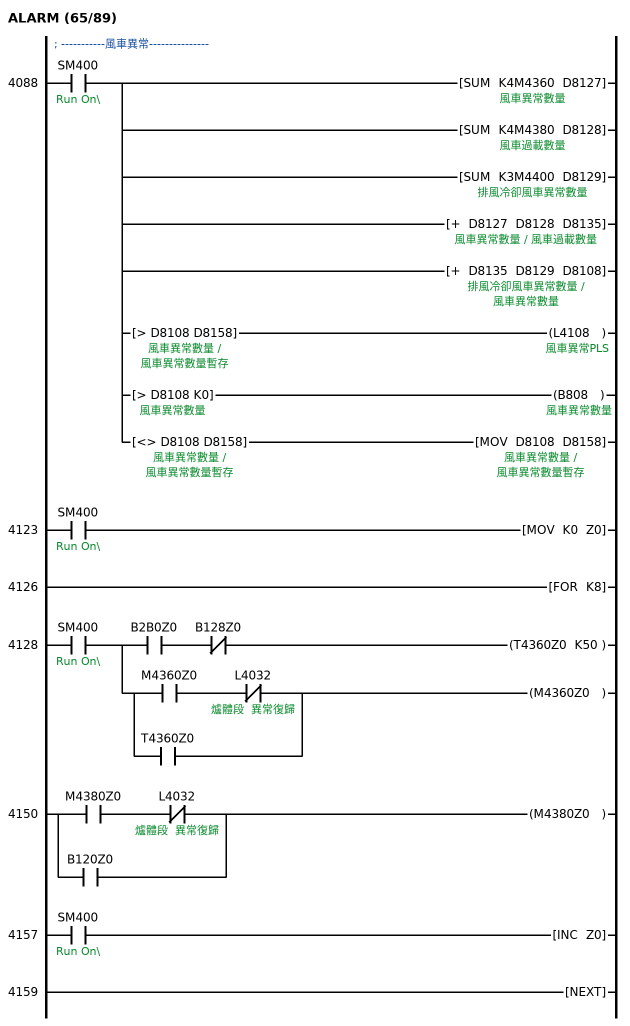
[picture p240: ladder of ALARM, rungs at steps 4088 to 4159]
; -----------風車異常---------------
4088  LD      SM400  ; Run On\
      SUM     K4M4360 D8127  ; 第01槽  風車馬達異常 / 風車異常數量
      SUM     K4M4380 D8128  ; 第01槽  風車馬達過載 / 風車過載數量
      SUM     K3M4400 D8129  ; 進料輸送排氣風車異常 / 排風冷卻風車異常數量
      +       D8127 D8128 D8135
      +       D8135 D8129 D8108  ; 風車異常數量
      MPS
      AND>    D8108 D8158  ; 風車異常數量 / 風車異常數量暫存
      OUT     L4108  ; 風車異常PLS
      MRD
      AND>    D8108 K0  ; 風車異常數量
      OUT     B808  ; 風車異常數量
      MPP
      AND<>   D8108 D8158  ; 風車異常數量 / 風車異常數量暫存
      MOV     D8108 D8158
4123  LD      SM400  ; Run On\
      MOV     K0 Z0
4126  FOR     K8
4128  LD      SM400  ; Run On\
      MPS
      AND     B2B0Z0
      ANI     B128Z0
      OUT     T4360Z0 K50
      MPP
      LD      M4360Z0
      ANI     L4032  ; 爐體段  異常復歸
      OR      T4360Z0
      ANB
      OUT     M4360Z0
4150  LD      M4380Z0
      ANI     L4032  ; 爐體段  異常復歸
      OR      B120Z0
      OUT     M4380Z0
4157  LD      SM400  ; Run On\
      INC     Z0
4159  NEXT
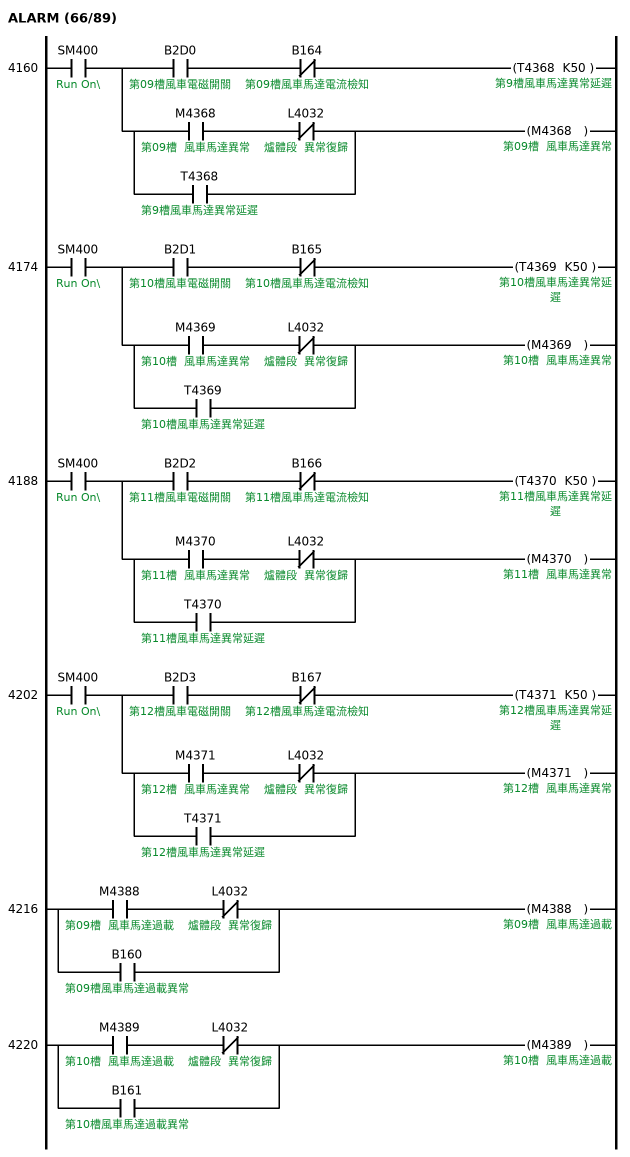
4160  LD      SM400  ; Run On\
      MPS
      AND     B2D0  ; 第09槽風車電磁開關
      ANI     B164  ; 第09槽風車馬達電流檢知
      OUT     T4368 K50  ; 第9槽風車馬達異常延遲
      MPP
      LD      M4368  ; 第09槽  風車馬達異常
      ANI     L4032  ; 爐體段  異常復歸
      OR      T4368  ; 第9槽風車馬達異常延遲
      ANB
      OUT     M4368  ; 第09槽  風車馬達異常
4174  LD      SM400  ; Run On\
      MPS
      AND     B2D1  ; 第10槽風車電磁開關
      ANI     B165  ; 第10槽風車馬達電流檢知
      OUT     T4369 K50  ; 第10槽風車馬達異常延遲
      MPP
      LD      M4369  ; 第10槽  風車馬達異常
      ANI     L4032  ; 爐體段  異常復歸
      OR      T4369  ; 第10槽風車馬達異常延遲
      ANB
      OUT     M4369  ; 第10槽  風車馬達異常
4188  LD      SM400  ; Run On\
      MPS
      AND     B2D2  ; 第11槽風車電磁開關
      ANI     B166  ; 第11槽風車馬達電流檢知
      OUT     T4370 K50  ; 第11槽風車馬達異常延遲
      MPP
      LD      M4370  ; 第11槽  風車馬達異常
      ANI     L4032  ; 爐體段  異常復歸
      OR      T4370  ; 第11槽風車馬達異常延遲
      ANB
      OUT     M4370  ; 第11槽  風車馬達異常
4202  LD      SM400  ; Run On\
      MPS
      AND     B2D3  ; 第12槽風車電磁開關
      ANI     B167  ; 第12槽風車馬達電流檢知
      OUT     T4371 K50  ; 第12槽風車馬達異常延遲
      MPP
      LD      M4371  ; 第12槽  風車馬達異常
      ANI     L4032  ; 爐體段  異常復歸
      OR      T4371  ; 第12槽風車馬達異常延遲
      ANB
      OUT     M4371  ; 第12槽  風車馬達異常
4216  LD      M4388  ; 第09槽  風車馬達過載
      ANI     L4032  ; 爐體段  異常復歸
      OR      B160  ; 第09槽風車馬達過載異常
      OUT     M4388  ; 第09槽  風車馬達過載
4220  LD      M4389  ; 第10槽  風車馬達過載
      ANI     L4032  ; 爐體段  異常復歸
      OR      B161  ; 第10槽風車馬達過載異常
      OUT     M4389  ; 第10槽  風車馬達過載
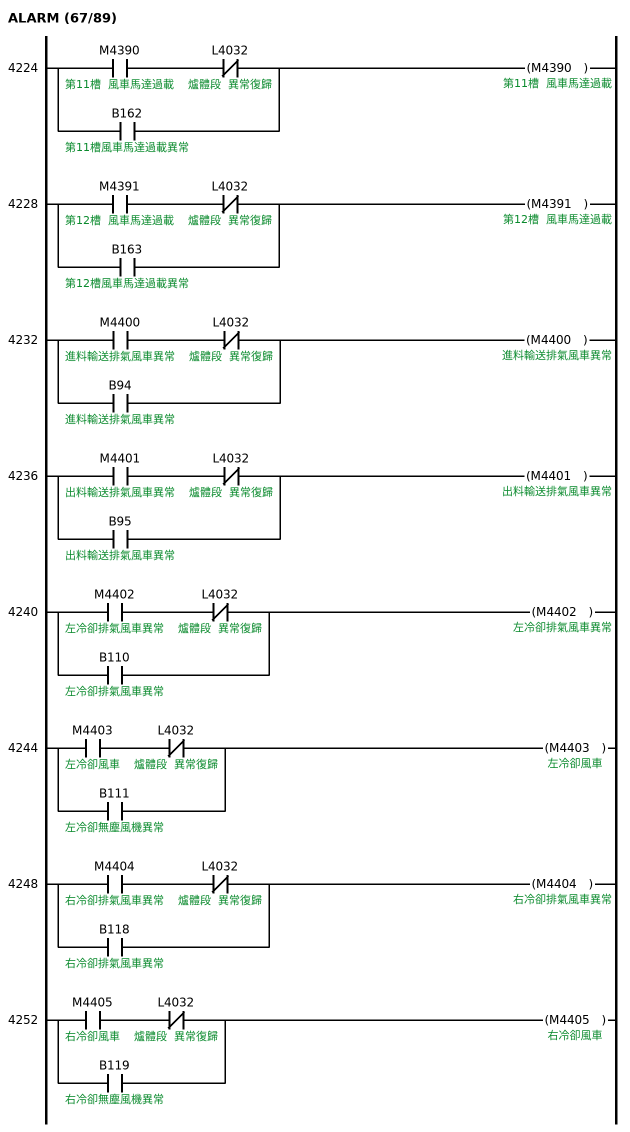
4224  LD      M4390  ; 第11槽  風車馬達過載
      ANI     L4032  ; 爐體段  異常復歸
      OR      B162  ; 第11槽風車馬達過載異常
      OUT     M4390  ; 第11槽  風車馬達過載
4228  LD      M4391  ; 第12槽  風車馬達過載
      ANI     L4032  ; 爐體段  異常復歸
      OR      B163  ; 第12槽風車馬達過載異常
      OUT     M4391  ; 第12槽  風車馬達過載
4232  LD      M4400  ; 進料輸送排氣風車異常
      ANI     L4032  ; 爐體段  異常復歸
      OR      B94  ; 進料輸送排氣風車異常
      OUT     M4400  ; 進料輸送排氣風車異常
4236  LD      M4401  ; 出料輸送排氣風車異常
      ANI     L4032  ; 爐體段  異常復歸
      OR      B95  ; 出料輸送排氣風車異常
      OUT     M4401  ; 出料輸送排氣風車異常
4240  LD      M4402  ; 左冷卻排氣風車異常
      ANI     L4032  ; 爐體段  異常復歸
      OR      B110  ; 左冷卻排氣風車異常
      OUT     M4402  ; 左冷卻排氣風車異常
4244  LD      M4403  ; 左冷卻風車
      ANI     L4032  ; 爐體段  異常復歸
      OR      B111  ; 左冷卻無塵風機異常
      OUT     M4403  ; 左冷卻風車
4248  LD      M4404  ; 右冷卻排氣風車異常
      ANI     L4032  ; 爐體段  異常復歸
      OR      B118  ; 右冷卻排氣風車異常
      OUT     M4404  ; 右冷卻排氣風車異常
4252  LD      M4405  ; 右冷卻風車
      ANI     L4032  ; 爐體段  異常復歸
      OR      B119  ; 右冷卻無塵風機異常
      OUT     M4405  ; 右冷卻風車
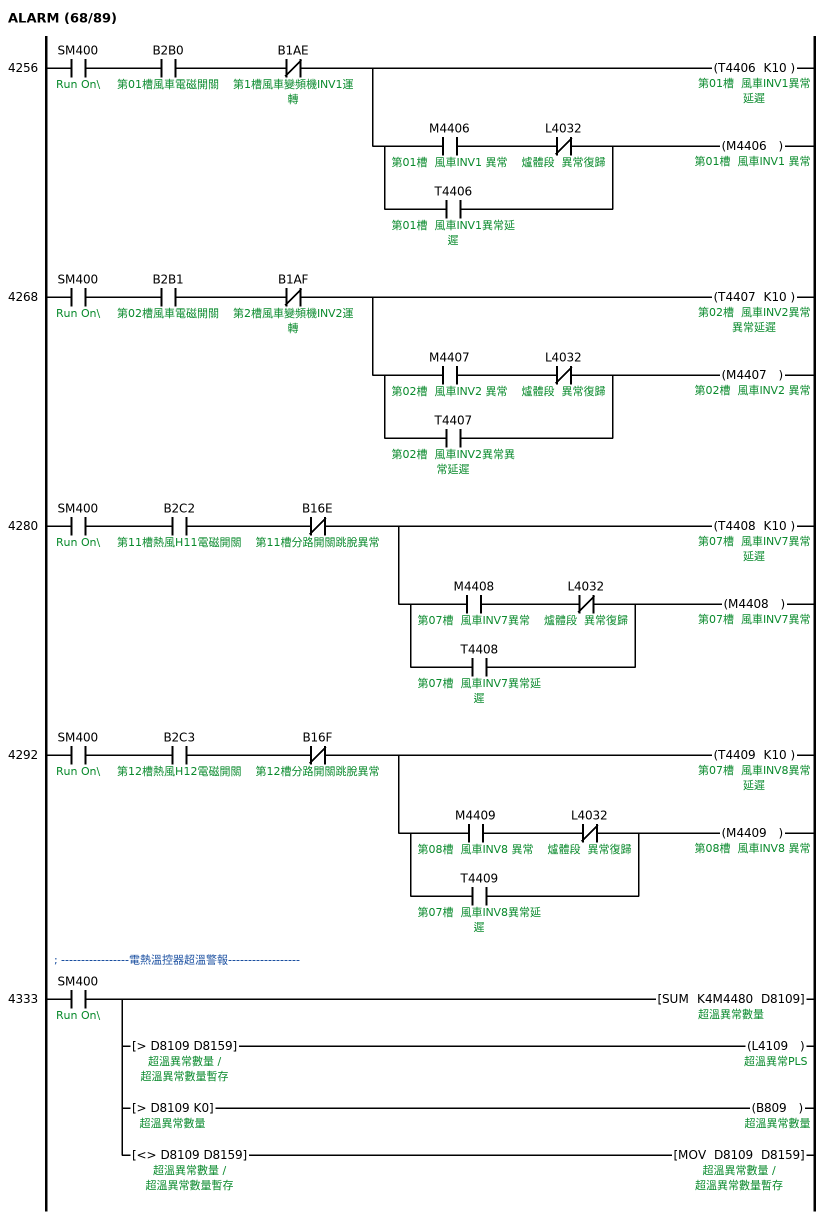
4256  LD      SM400  ; Run On\
      AND     B2B0  ; 第01槽風車電磁開關
      ANI     B1AE  ; 第1槽風車變頻機INV1運轉
      OUT     T4406 K10  ; 第01槽  風車INV1異常延遲
      LD      M4406  ; 第01槽  風車INV1 異常
      ANI     L4032  ; 爐體段  異常復歸
      OR      T4406  ; 第01槽  風車INV1異常延遲
      ANB
      OUT     M4406  ; 第01槽  風車INV1 異常
4268  LD      SM400  ; Run On\
      AND     B2B1  ; 第02槽風車電磁開關
      ANI     B1AF  ; 第2槽風車變頻機INV2運轉
      OUT     T4407 K10  ; 第02槽  風車INV2異常異常延遲
      LD      M4407  ; 第02槽  風車INV2 異常
      ANI     L4032  ; 爐體段  異常復歸
      OR      T4407  ; 第02槽  風車INV2異常異常延遲
      ANB
      OUT     M4407  ; 第02槽  風車INV2 異常
4280  LD      SM400  ; Run On\
      AND     B2C2  ; 第11槽熱風H11電磁開關
      ANI     B16E  ; 第11槽分路開關跳脫異常
      OUT     T4408 K10  ; 第07槽  風車INV7異常延遲
      LD      M4408  ; 第07槽  風車INV7異常
      ANI     L4032  ; 爐體段  異常復歸
      OR      T4408  ; 第07槽  風車INV7異常延遲
      ANB
      OUT     M4408  ; 第07槽  風車INV7異常
4292  LD      SM400  ; Run On\
      AND     B2C3  ; 第12槽熱風H12電磁開關
      ANI     B16F  ; 第12槽分路開關跳脫異常
      OUT     T4409 K10  ; 第07槽  風車INV8異常延遲
      LD      M4409  ; 第08槽  風車INV8 異常
      ANI     L4032  ; 爐體段  異常復歸
      OR      T4409  ; 第07槽  風車INV8異常延遲
      ANB
      OUT     M4409  ; 第08槽  風車INV8 異常
; -----------------電熱溫控器超溫警報------------------
4333  LD      SM400  ; Run On\
      SUM     K4M4480 D8109  ; 第01槽 熱風超溫異常 / 超溫異常數量
      MPS
      AND>    D8109 D8159  ; 超溫異常數量 / 超溫異常數量暫存
      OUT     L4109  ; 超溫異常PLS
      MRD
      AND>    D8109 K0  ; 超溫異常數量
      OUT     B809  ; 超溫異常數量
      MPP
      AND<>   D8109 D8159  ; 超溫異常數量 / 超溫異常數量暫存
      MOV     D8109 D8159
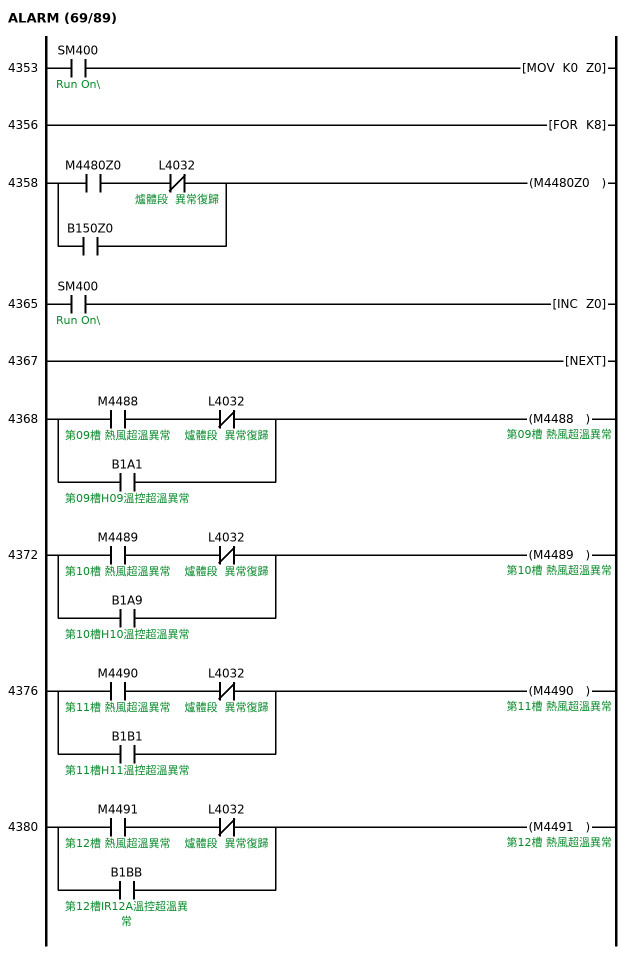
4353  LD      SM400  ; Run On\
      MOV     K0 Z0
4356  FOR     K8
4358  LD      M4480Z0
      ANI     L4032  ; 爐體段  異常復歸
      OR      B150Z0
      OUT     M4480Z0
4365  LD      SM400  ; Run On\
      INC     Z0
4367  NEXT
4368  LD      M4488  ; 第09槽 熱風超溫異常
      ANI     L4032  ; 爐體段  異常復歸
      OR      B1A1  ; 第09槽H09溫控超溫異常
      OUT     M4488  ; 第09槽 熱風超溫異常
4372  LD      M4489  ; 第10槽 熱風超溫異常
      ANI     L4032  ; 爐體段  異常復歸
      OR      B1A9  ; 第10槽H10溫控超溫異常
      OUT     M4489  ; 第10槽 熱風超溫異常
4376  LD      M4490  ; 第11槽 熱風超溫異常
      ANI     L4032  ; 爐體段  異常復歸
      OR      B1B1  ; 第11槽H11溫控超溫異常
      OUT     M4490  ; 第11槽 熱風超溫異常
4380  LD      M4491  ; 第12槽 熱風超溫異常
      ANI     L4032  ; 爐體段  異常復歸
      OR      B1BB  ; 第12槽IR12A溫控超溫異常
      OUT     M4491  ; 第12槽 熱風超溫異常
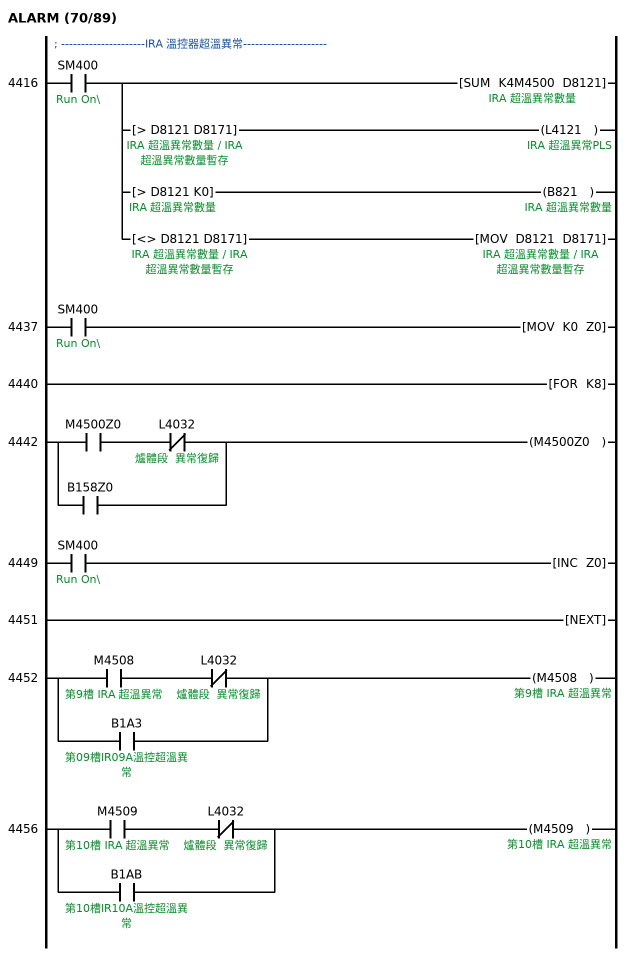
; ---------------------IRA 溫控器超溫異常---------------------
4416  LD      SM400  ; Run On\
      SUM     K4M4500 D8121  ; 第1槽 IRA 超溫異常 / IRA 超溫異常數量
      MPS
      AND>    D8121 D8171  ; IRA 超溫異常數量 / IRA 超溫異常數量暫存
      OUT     L4121  ; IRA 超溫異常PLS
      MRD
      AND>    D8121 K0  ; IRA 超溫異常數量
      OUT     B821  ; IRA 超溫異常數量
      MPP
      AND<>   D8121 D8171  ; IRA 超溫異常數量 / IRA 超溫異常數量暫存
      MOV     D8121 D8171
4437  LD      SM400  ; Run On\
      MOV     K0 Z0
4440  FOR     K8
4442  LD      M4500Z0
      ANI     L4032  ; 爐體段  異常復歸
      OR      B158Z0
      OUT     M4500Z0
4449  LD      SM400  ; Run On\
      INC     Z0
4451  NEXT
4452  LD      M4508  ; 第9槽 IRA 超溫異常
      ANI     L4032  ; 爐體段  異常復歸
      OR      B1A3  ; 第09槽IR09A溫控超溫異常
      OUT     M4508  ; 第9槽 IRA 超溫異常
4456  LD      M4509  ; 第10槽 IRA 超溫異常
      ANI     L4032  ; 爐體段  異常復歸
      OR      B1AB  ; 第10槽IR10A溫控超溫異常
      OUT     M4509  ; 第10槽 IRA 超溫異常
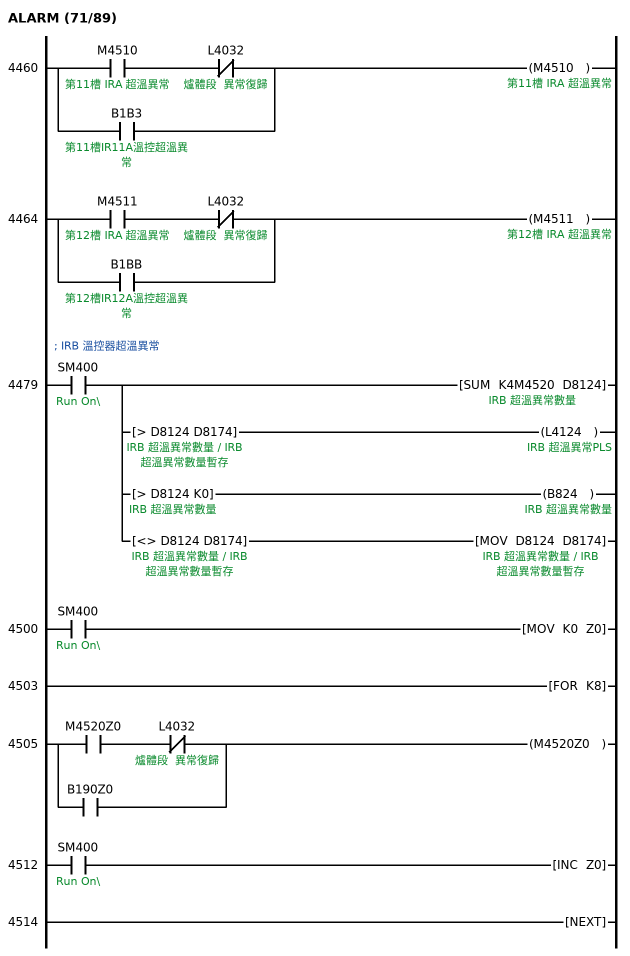
4460  LD      M4510  ; 第11槽 IRA 超溫異常
      ANI     L4032  ; 爐體段  異常復歸
      OR      B1B3  ; 第11槽IR11A溫控超溫異常
      OUT     M4510  ; 第11槽 IRA 超溫異常
4464  LD      M4511  ; 第12槽 IRA 超溫異常
      ANI     L4032  ; 爐體段  異常復歸
      OR      B1BB  ; 第12槽IR12A溫控超溫異常
      OUT     M4511  ; 第12槽 IRA 超溫異常
; IRB 溫控器超溫異常
4479  LD      SM400  ; Run On\
      SUM     K4M4520 D8124  ; 第1槽 IRB 超溫異常 / IRB 超溫異常數量
      MPS
      AND>    D8124 D8174  ; IRB 超溫異常數量 / IRB 超溫異常數量暫存
      OUT     L4124  ; IRB 超溫異常PLS
      MRD
      AND>    D8124 K0  ; IRB 超溫異常數量
      OUT     B824  ; IRB 超溫異常數量
      MPP
      AND<>   D8124 D8174  ; IRB 超溫異常數量 / IRB 超溫異常數量暫存
      MOV     D8124 D8174
4500  LD      SM400  ; Run On\
      MOV     K0 Z0
4503  FOR     K8
4505  LD      M4520Z0
      ANI     L4032  ; 爐體段  異常復歸
      OR      B190Z0
      OUT     M4520Z0
4512  LD      SM400  ; Run On\
      INC     Z0
4514  NEXT
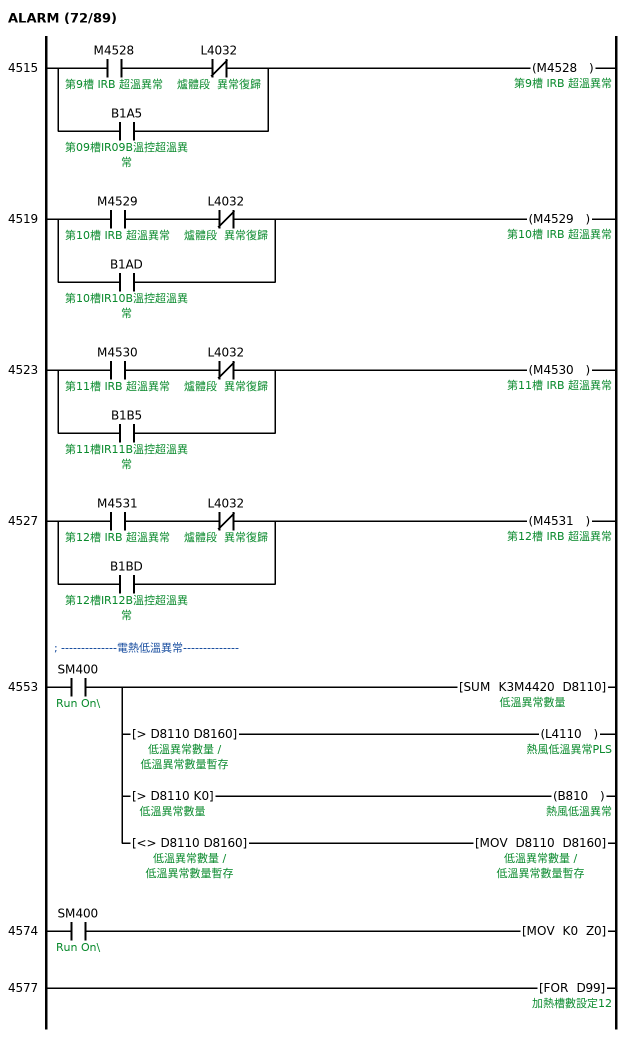
4515  LD      M4528  ; 第9槽 IRB 超溫異常
      ANI     L4032  ; 爐體段  異常復歸
      OR      B1A5  ; 第09槽IR09B溫控超溫異常
      OUT     M4528  ; 第9槽 IRB 超溫異常
4519  LD      M4529  ; 第10槽 IRB 超溫異常
      ANI     L4032  ; 爐體段  異常復歸
      OR      B1AD  ; 第10槽IR10B溫控超溫異常
      OUT     M4529  ; 第10槽 IRB 超溫異常
4523  LD      M4530  ; 第11槽 IRB 超溫異常
      ANI     L4032  ; 爐體段  異常復歸
      OR      B1B5  ; 第11槽IR11B溫控超溫異常
      OUT     M4530  ; 第11槽 IRB 超溫異常
4527  LD      M4531  ; 第12槽 IRB 超溫異常
      ANI     L4032  ; 爐體段  異常復歸
      OR      B1BD  ; 第12槽IR12B溫控超溫異常
      OUT     M4531  ; 第12槽 IRB 超溫異常
; --------------電熱低溫異常--------------
4553  LD      SM400  ; Run On\
      SUM     K3M4420 D8110  ; 第01槽 熱風低溫異常 / 低溫異常數量
      MPS
      AND>    D8110 D8160  ; 低溫異常數量 / 低溫異常數量暫存
      OUT     L4110  ; 熱風低溫異常PLS
      MRD
      AND>    D8110 K0  ; 低溫異常數量
      OUT     B810  ; 熱風低溫異常
      MPP
      AND<>   D8110 D8160  ; 低溫異常數量 / 低溫異常數量暫存
      MOV     D8110 D8160
4574  LD      SM400  ; Run On\
      MOV     K0 Z0
4577  FOR     D99  ; 加熱槽數設定12
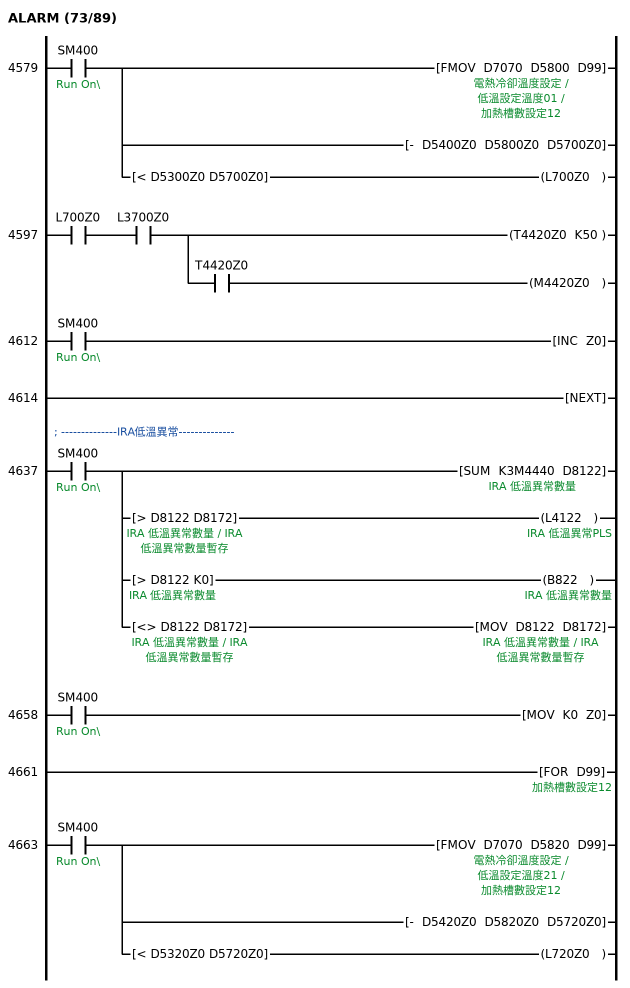
4579  LD      SM400  ; Run On\
      FMOV    D7070 D5800 D99  ; 電熱冷卻溫度設定 / 低溫設定溫度01
      -       D5400Z0 D5800Z0 D5700Z0
      AND<    D5300Z0 D5700Z0
      OUT     L700Z0
4597  LD      L700Z0
      AND     L3700Z0
      OUT     T4420Z0 K50
      AND     T4420Z0
      OUT     M4420Z0
4612  LD      SM400  ; Run On\
      INC     Z0
4614  NEXT
; --------------IRA低溫異常--------------
4637  LD      SM400  ; Run On\
      SUM     K3M4440 D8122  ; 第01槽 IRA 低溫異常 / IRA 低溫異常數量
      MPS
      AND>    D8122 D8172  ; IRA 低溫異常數量 / IRA 低溫異常數量暫存
      OUT     L4122  ; IRA 低溫異常PLS
      MRD
      AND>    D8122 K0  ; IRA 低溫異常數量
      OUT     B822  ; IRA 低溫異常數量
      MPP
      AND<>   D8122 D8172  ; IRA 低溫異常數量 / IRA 低溫異常數量暫存
      MOV     D8122 D8172
4658  LD      SM400  ; Run On\
      MOV     K0 Z0
4661  FOR     D99
4663  LD      SM400  ; Run On\
      FMOV    D7070 D5820 D99  ; 低溫設定溫度21
      -       D5420Z0 D5820Z0 D5720Z0
      AND<    D5320Z0 D5720Z0
      OUT     L720Z0
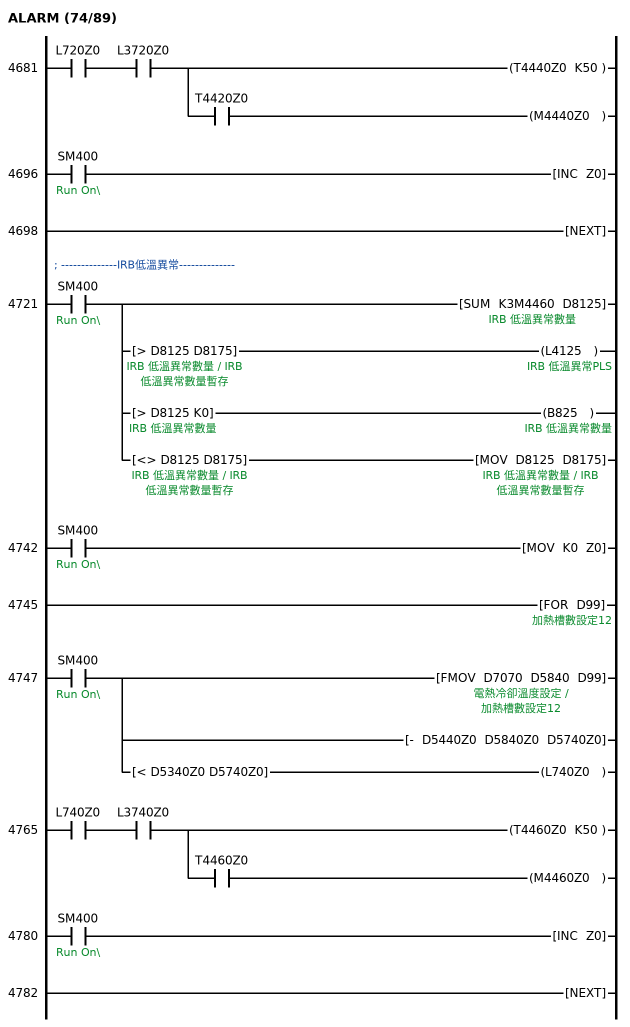
4681  LD      L720Z0
      AND     L3720Z0
      OUT     T4440Z0 K50
      AND     T4420Z0
      OUT     M4440Z0
4696  LD      SM400  ; Run On\
      INC     Z0
4698  NEXT
; --------------IRB低溫異常--------------
4721  LD      SM400  ; Run On\
      SUM     K3M4460 D8125  ; 第01槽 IRB 低溫異常 / IRB 低溫異常數量
      MPS
      AND>    D8125 D8175  ; IRB 低溫異常數量 / IRB 低溫異常數量暫存
      OUT     L4125  ; IRB 低溫異常PLS
      MRD
      AND>    D8125 K0  ; IRB 低溫異常數量
      OUT     B825  ; IRB 低溫異常數量
      MPP
      AND<>   D8125 D8175  ; IRB 低溫異常數量 / IRB 低溫異常數量暫存
      MOV     D8125 D8175
4742  LD      SM400  ; Run On\
      MOV     K0 Z0
4745  FOR     D99
4747  LD      SM400  ; Run On\
      FMOV    D7070 D5840 D99
      -       D5440Z0 D5840Z0 D5740Z0
      AND<    D5340Z0 D5740Z0
      OUT     L740Z0
4765  LD      L740Z0
      AND     L3740Z0
      OUT     T4460Z0 K50
      AND     T4460Z0
      OUT     M4460Z0
4780  LD      SM400  ; Run On\
      INC     Z0
4782  NEXT
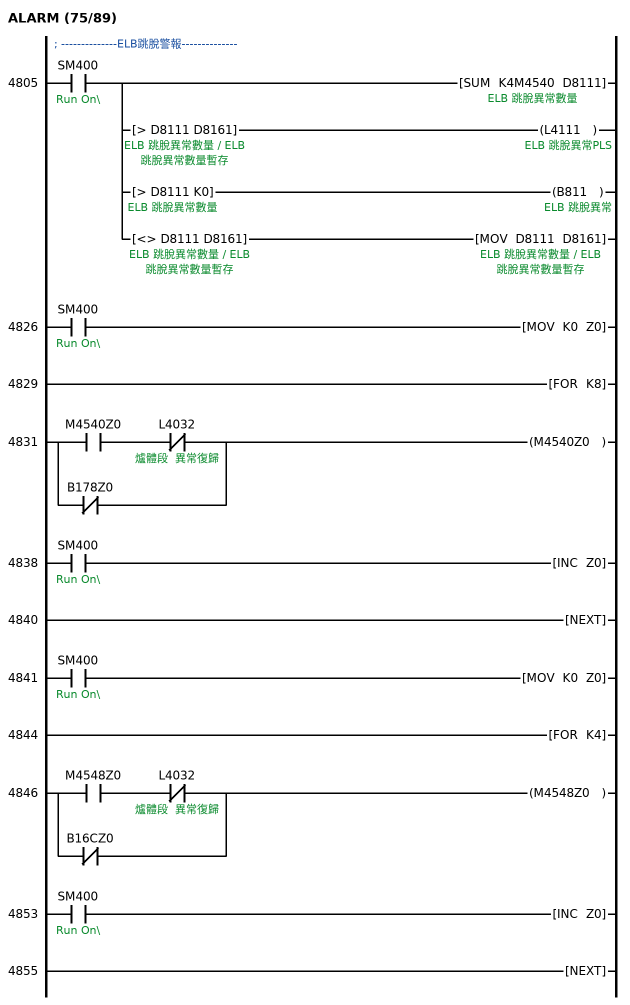
; --------------ELB跳脫警報--------------
4805  LD      SM400  ; Run On\
      SUM     K4M4540 D8111  ; 第01槽  分路開關跳脫異常 / ELB 跳脫異常數量
      MPS
      AND>    D8111 D8161  ; ELB 跳脫異常數量 / ELB 跳脫異常數量暫存
      OUT     L4111  ; ELB 跳脫異常PLS
      MRD
      AND>    D8111 K0  ; ELB 跳脫異常數量
      OUT     B811  ; ELB 跳脫異常
      MPP
      AND<>   D8111 D8161  ; ELB 跳脫異常數量 / ELB 跳脫異常數量暫存
      MOV     D8111 D8161
4826  LD      SM400  ; Run On\
      MOV     K0 Z0
4829  FOR     K8
4831  LD      M4540Z0
      ANI     L4032  ; 爐體段  異常復歸
      ORI     B178Z0
      OUT     M4540Z0
4838  LD      SM400  ; Run On\
      INC     Z0
4840  NEXT
4841  LD      SM400  ; Run On\
      MOV     K0 Z0
4844  FOR     K4
4846  LD      M4548Z0
      ANI     L4032  ; 爐體段  異常復歸
      ORI     B16CZ0
      OUT     M4548Z0
4853  LD      SM400  ; Run On\
      INC     Z0
4855  NEXT
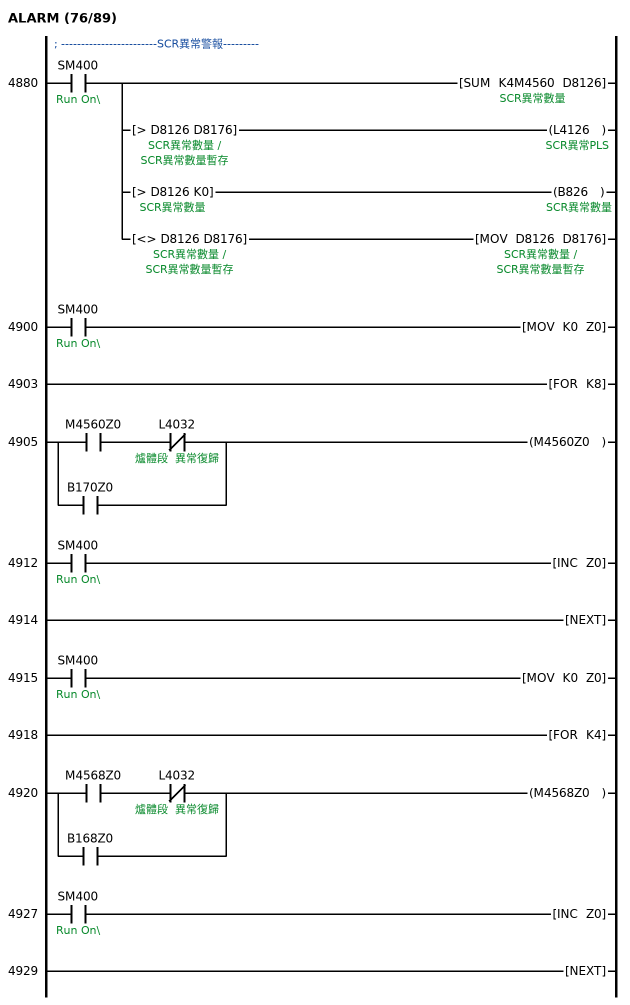
; ------------------------SCR異常警報---------
4880  LD      SM400  ; Run On\
      SUM     K4M4560 D8126  ; 第01槽  SCR異常 / SCR異常數量
      MPS
      AND>    D8126 D8176  ; SCR異常數量 / SCR異常數量暫存
      OUT     L4126  ; SCR異常PLS
      MRD
      AND>    D8126 K0  ; SCR異常數量
      OUT     B826  ; SCR異常數量
      MPP
      AND<>   D8126 D8176  ; SCR異常數量 / SCR異常數量暫存
      MOV     D8126 D8176
4900  LD      SM400  ; Run On\
      MOV     K0 Z0
4903  FOR     K8
4905  LD      M4560Z0
      ANI     L4032  ; 爐體段  異常復歸
      OR      B170Z0
      OUT     M4560Z0
4912  LD      SM400  ; Run On\
      INC     Z0
4914  NEXT
4915  LD      SM400  ; Run On\
      MOV     K0 Z0
4918  FOR     K4
4920  LD      M4568Z0
      ANI     L4032  ; 爐體段  異常復歸
      OR      B168Z0
      OUT     M4568Z0
4927  LD      SM400  ; Run On\
      INC     Z0
4929  NEXT
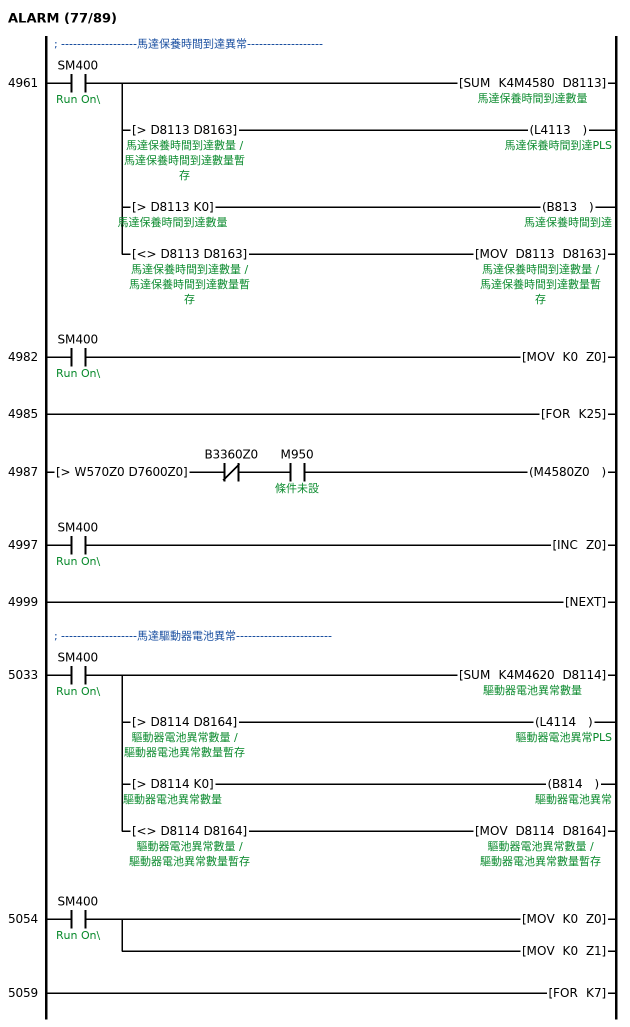
; -------------------馬達保養時間到達異常-------------------
4961  LD      SM400  ; Run On\
      SUM     K4M4580 D8113  ; 馬達保養時間到達數量
      MPS
      AND>    D8113 D8163  ; 馬達保養時間到達數量 / 馬達保養時間到達數量暫存
      OUT     L4113  ; 馬達保養時間到達PLS
      MRD
      AND>    D8113 K0  ; 馬達保養時間到達數量
      OUT     B813  ; 馬達保養時間到達
      MPP
      AND<>   D8113 D8163  ; 馬達保養時間到達數量 / 馬達保養時間到達數量暫存
      MOV     D8113 D8163
4982  LD      SM400  ; Run On\
      MOV     K0 Z0
4985  FOR     K25
4987  LD>     W570Z0 D7600Z0
      ANI     B3360Z0
      AND     M950  ; 條件未設
      OUT     M4580Z0
4997  LD      SM400  ; Run On\
      INC     Z0
4999  NEXT
; -------------------馬達驅動器電池異常------------------------
5033  LD      SM400  ; Run On\
      SUM     K4M4620 D8114  ; 進料整板驅動器電池異常 / 驅動器電池異常數量
      MPS
      AND>    D8114 D8164  ; 驅動器電池異常數量 / 驅動器電池異常數量暫存
      OUT     L4114  ; 驅動器電池異常PLS
      MRD
      AND>    D8114 K0  ; 驅動器電池異常數量
      OUT     B814  ; 驅動器電池異常
      MPP
      AND<>   D8114 D8164  ; 驅動器電池異常數量 / 驅動器電池異常數量暫存
      MOV     D8114 D8164
5054  LD      SM400  ; Run On\
      MOV     K0 Z0
      MOV     K0 Z1
5059  FOR     K7
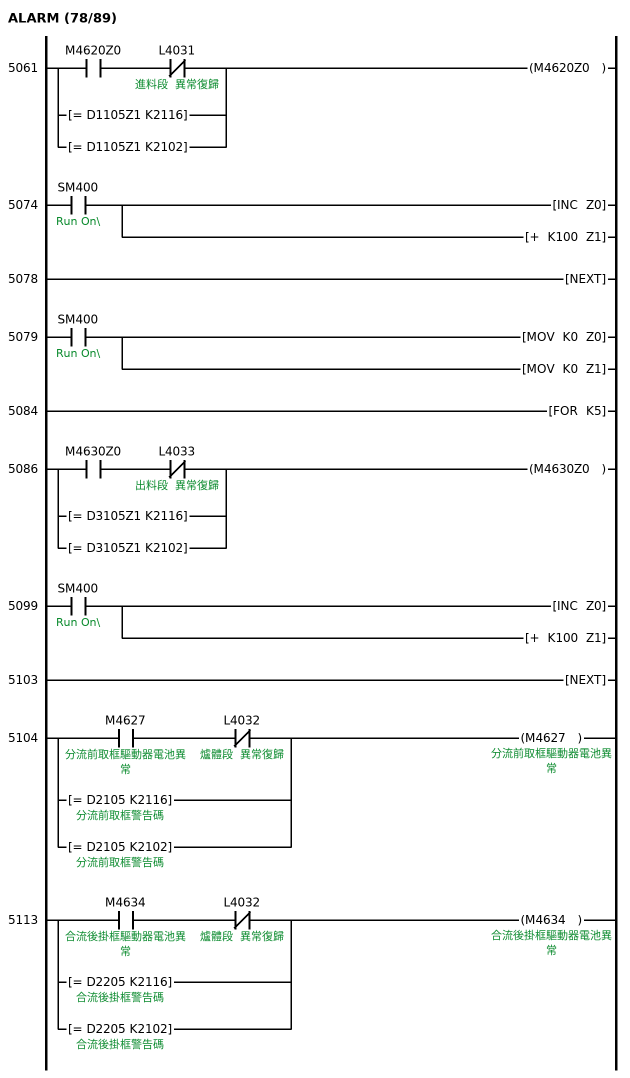
5061  LD      M4620Z0
      ANI     L4031  ; 進料段  異常復歸
      OR=     D1105Z1 K2116
      OR=     D1105Z1 K2102
      OUT     M4620Z0
5074  LD      SM400  ; Run On\
      INC     Z0
      +       K100 Z1
5078  NEXT
5079  LD      SM400  ; Run On\
      MOV     K0 Z0
      MOV     K0 Z1
5084  FOR     K5
5086  LD      M4630Z0
      ANI     L4033  ; 出料段  異常復歸
      OR=     D3105Z1 K2116
      OR=     D3105Z1 K2102
      OUT     M4630Z0
5099  LD      SM400  ; Run On\
      INC     Z0
      +       K100 Z1
5103  NEXT
5104  LD      M4627  ; 分流前取框驅動器電池異常
      ANI     L4032  ; 爐體段  異常復歸
      OR=     D2105 K2116  ; 分流前取框警告碼
      OR=     D2105 K2102  ; 分流前取框警告碼
      OUT     M4627  ; 分流前取框驅動器電池異常
5113  LD      M4634  ; 合流後掛框驅動器電池異常
      ANI     L4032  ; 爐體段  異常復歸
      OR=     D2205 K2116  ; 合流後掛框警告碼
      OR=     D2205 K2102  ; 合流後掛框警告碼
      OUT     M4634  ; 合流後掛框驅動器電池異常
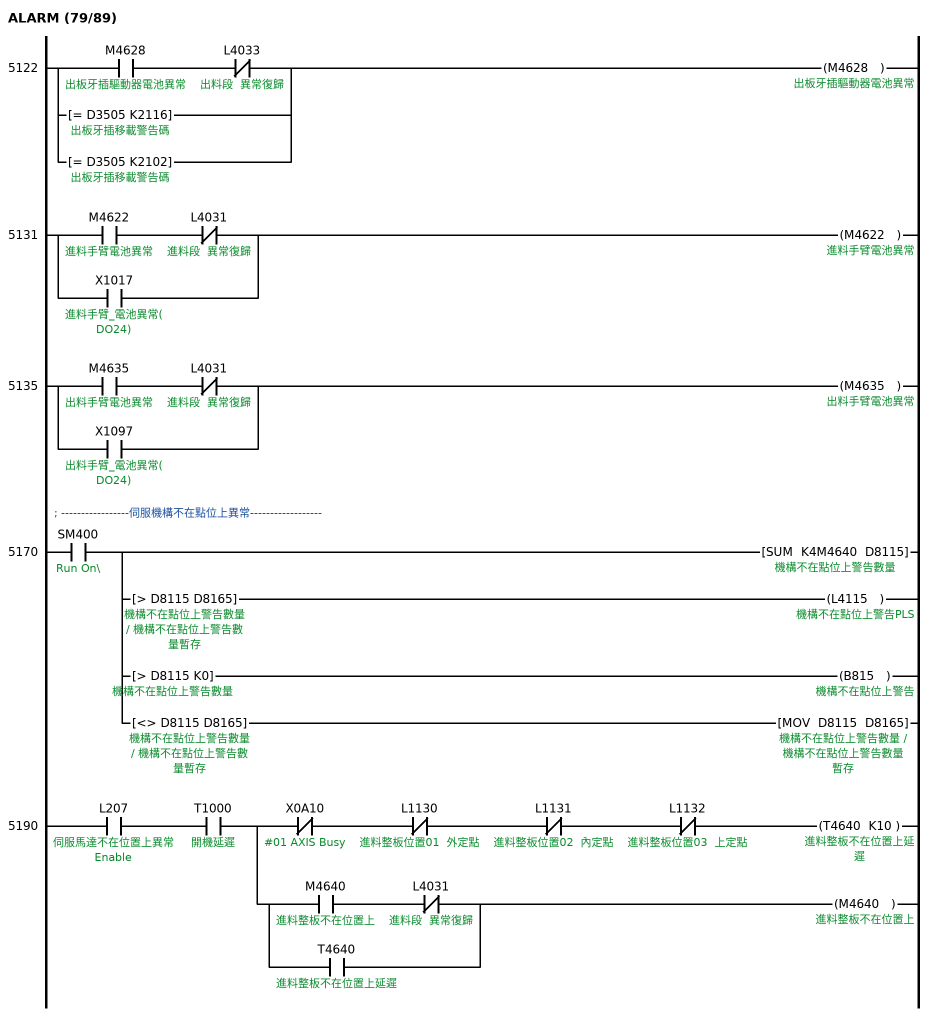
5122  LD      M4628  ; 出板牙插驅動器電池異常
      ANI     L4033  ; 出料段  異常復歸
      OR=     D3505 K2116  ; 出板牙插移載警告碼
      OR=     D3505 K2102  ; 出板牙插移載警告碼
      OUT     M4628  ; 出板牙插驅動器電池異常
5131  LD      M4622  ; 進料手臂電池異常
      ANI     L4031  ; 進料段  異常復歸
      OR      X1017  ; 進料手臂_電池異常(DO24)
      OUT     M4622  ; 進料手臂電池異常
5135  LD      M4635  ; 出料手臂電池異常
      ANI     L4031  ; 進料段  異常復歸
      OR      X1097  ; 出料手臂_電池異常(DO24)
      OUT     M4635  ; 出料手臂電池異常
; -----------------伺服機構不在點位上異常------------------
5170  LD      SM400  ; Run On\
      SUM     K4M4640 D8115  ; 進料整板不在位置上 / 機構不在點位上警告數量
      MPS
      AND>    D8115 D8165  ; 機構不在點位上警告數量 / 機構不在點位上警告數量暫存
      OUT     L4115  ; 機構不在點位上警告PLS
      MRD
      AND>    D8115 K0  ; 機構不在點位上警告數量
      OUT     B815  ; 機構不在點位上警告
      MPP
      AND<>   D8115 D8165  ; 機構不在點位上警告數量 / 機構不在點位上警告數量暫存
      MOV     D8115 D8165
5190  LD      L207  ; 伺服馬達不在位置上異常  Enable
      AND     T1000  ; 開機延遲
      MPS
      ANI     X0A10  ; #01 AXIS Busy
      ANI     L1130  ; 進料整板位置01  外定點
      ANI     L1131  ; 進料整板位置02  內定點
      ANI     L1132  ; 進料整板位置03  上定點
      OUT     T4640 K10  ; 進料整板不在位置上延遲
      MPP
      LD      M4640  ; 進料整板不在位置上
      ANI     L4031  ; 進料段  異常復歸
      OR      T4640  ; 進料整板不在位置上延遲
      ANB
      OUT     M4640  ; 進料整板不在位置上
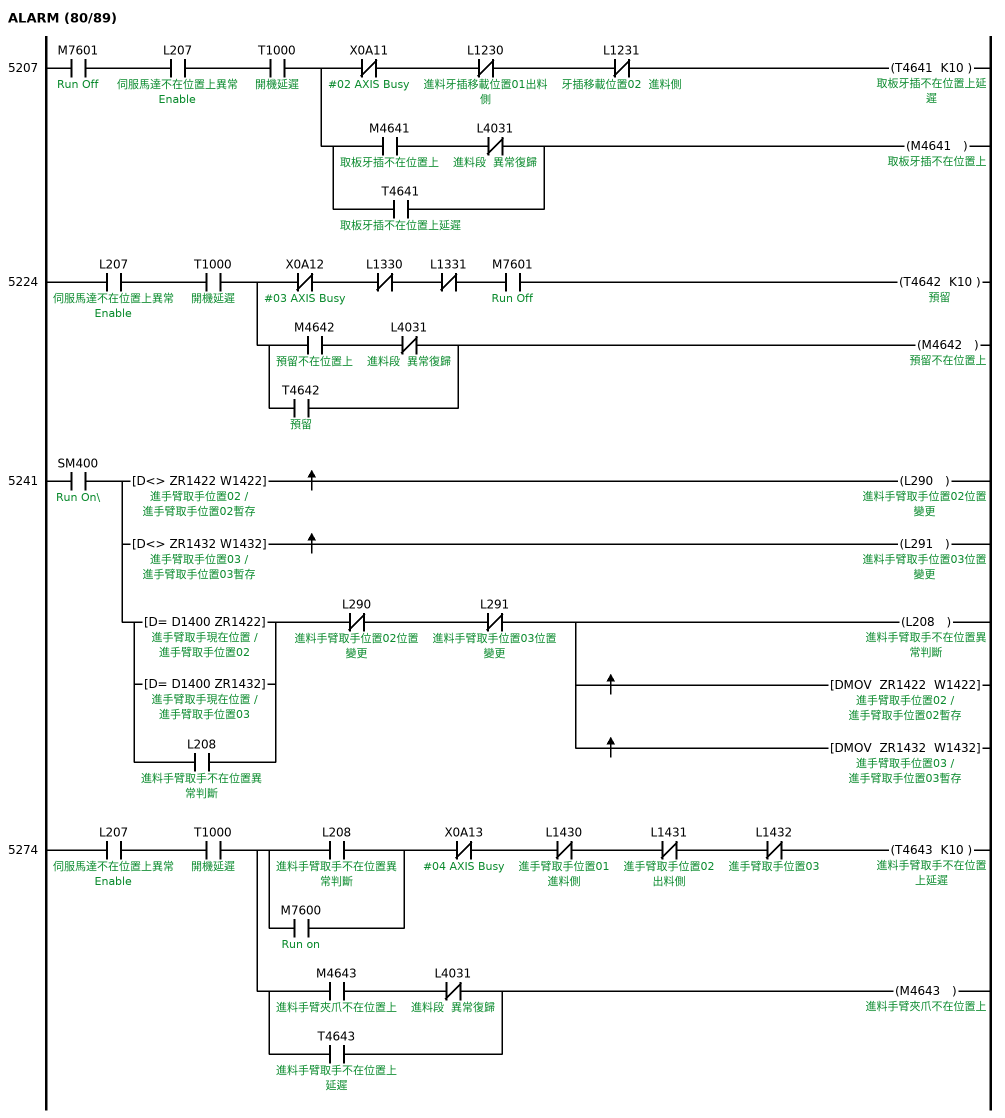
5207  LD      M7601  ; Run Off
      AND     L207  ; 伺服馬達不在位置上異常  Enable
      AND     T1000  ; 開機延遲
      MPS
      ANI     X0A11  ; #02 AXIS Busy
      ANI     L1230  ; 進料牙插移載位置01出料側
      ANI     L1231  ; 牙插移載位置02  進料側
      OUT     T4641 K10  ; 取板牙插不在位置上延遲
      MPP
      LD      M4641  ; 取板牙插不在位置上
      ANI     L4031  ; 進料段  異常復歸
      OR      T4641  ; 取板牙插不在位置上延遲
      ANB
      OUT     M4641  ; 取板牙插不在位置上
5224  LD      L207  ; 伺服馬達不在位置上異常  Enable
      AND     T1000  ; 開機延遲
      MPS
      ANI     X0A12  ; #03 AXIS Busy
      ANI     L1330
      ANI     L1331
      AND     M7601  ; Run Off
      OUT     T4642 K10  ; 預留
      MPP
      LD      M4642  ; 預留不在位置上
      ANI     L4031  ; 進料段  異常復歸
      OR      T4642  ; 預留
      ANB
      OUT     M4642  ; 預留不在位置上
5241  LD      SM400  ; Run On\
      MPS
      ANDD<>  ZR1422 W1422  ; 進手臂取手位置02 / 進手臂取手位置02暫存
      MEP
      OUT     L290  ; 進料手臂取手位置02位置變更
      MRD
      ANDD<>  ZR1432 W1432  ; 進手臂取手位置03 / 進手臂取手位置03暫存
      MEP
      OUT     L291  ; 進料手臂取手位置03位置變更
      MPP
      LDD=    D1400 ZR1422  ; 進手臂取手現在位置 / 進手臂取手位置02
      ORD=    D1400 ZR1432  ; 進手臂取手現在位置 / 進手臂取手位置03
      OR      L208  ; 進料手臂取手不在位置異常判斷
      ANB
      ANI     L290  ; 進料手臂取手位置02位置變更
      ANI     L291  ; 進料手臂取手位置03位置變更
      OUT     L208  ; 進料手臂取手不在位置異常判斷
      MPS
      MEP
      DMOV    ZR1422 W1422
      MPP
      MEP
      DMOV    ZR1432 W1432
5274  LD      L207  ; 伺服馬達不在位置上異常  Enable
      AND     T1000  ; 開機延遲
      MPS
      LD      L208  ; 進料手臂取手不在位置異常判斷
      OR      M7600  ; Run on
      ANB
      ANI     X0A13  ; #04 AXIS Busy
      ANI     L1430  ; 進手臂取手位置01  進料側
      ANI     L1431  ; 進手臂取手位置02  出料側
      ANI     L1432  ; 進手臂取手位置03
      OUT     T4643 K10  ; 進料手臂取手不在位置上延遲
      MPP
      LD      M4643  ; 進料手臂夾爪不在位置上
      ANI     L4031  ; 進料段  異常復歸
      OR      T4643  ; 進料手臂取手不在位置上延遲
      ANB
      OUT     M4643  ; 進料手臂夾爪不在位置上
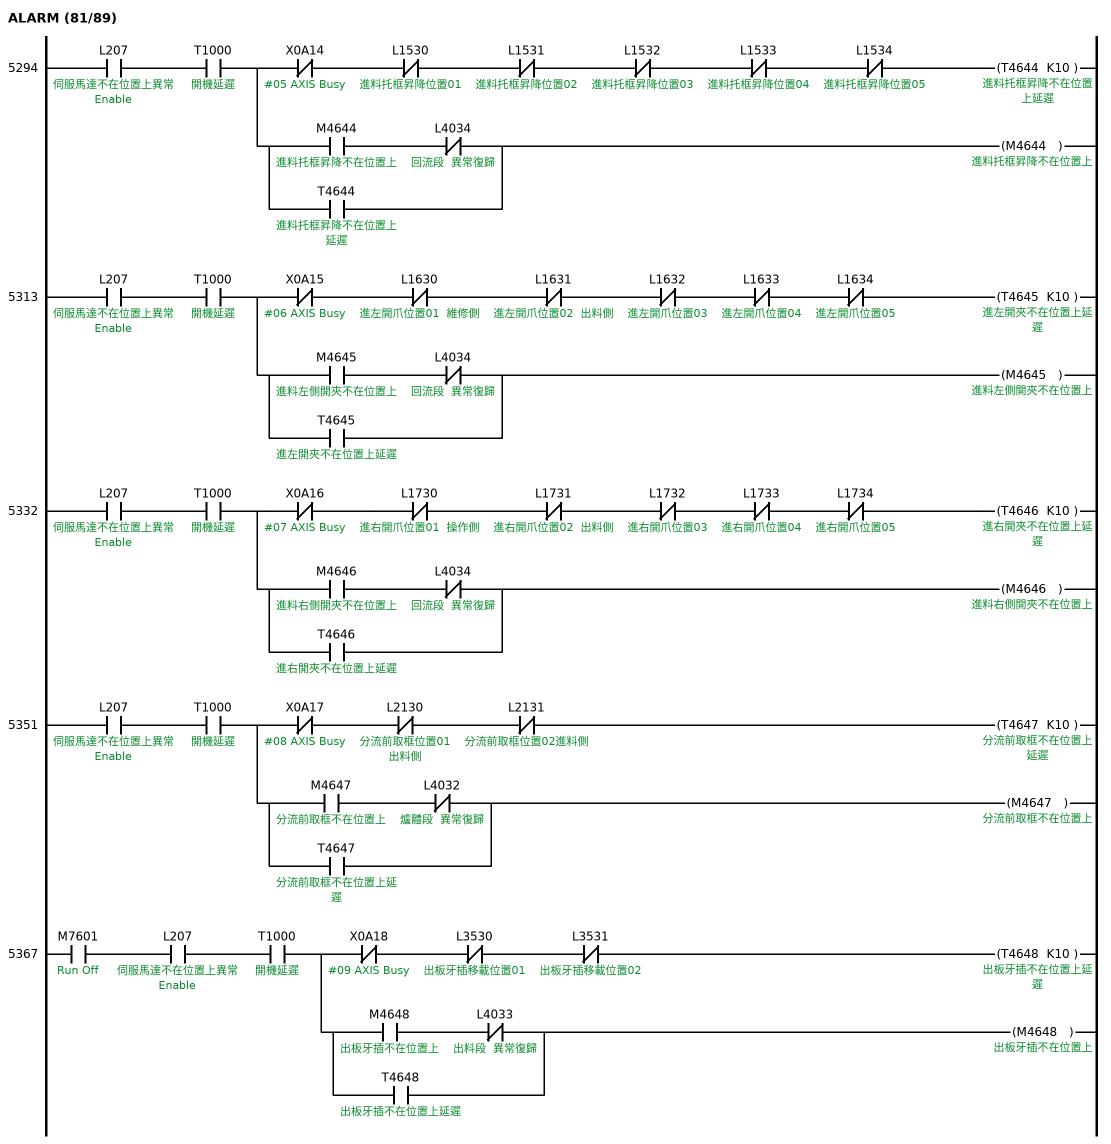
5294  LD      L207  ; 伺服馬達不在位置上異常  Enable
      AND     T1000  ; 開機延遲
      MPS
      ANI     X0A14  ; #05 AXIS Busy
      ANI     L1530  ; 進料托框昇降位置01
      ANI     L1531  ; 進料托框昇降位置02
      ANI     L1532  ; 進料托框昇降位置03
      ANI     L1533  ; 進料托框昇降位置04
      ANI     L1534  ; 進料托框昇降位置05
      OUT     T4644 K10  ; 進料托框昇降不在位置上延遲
      MPP
      LD      M4644  ; 進料托框昇降不在位置上
      ANI     L4034  ; 回流段  異常復歸
      OR      T4644  ; 進料托框昇降不在位置上延遲
      ANB
      OUT     M4644  ; 進料托框昇降不在位置上
5313  LD      L207  ; 伺服馬達不在位置上異常  Enable
      AND     T1000  ; 開機延遲
      MPS
      ANI     X0A15  ; #06 AXIS Busy
      ANI     L1630  ; 進左開爪位置01  維修側
      ANI     L1631  ; 進左開爪位置02  出料側
      ANI     L1632  ; 進左開爪位置03
      ANI     L1633  ; 進左開爪位置04
      ANI     L1634  ; 進左開爪位置05
      OUT     T4645 K10  ; 進左開夾不在位置上延遲
      MPP
      LD      M4645  ; 進料左側開夾不在位置上
      ANI     L4034  ; 回流段  異常復歸
      OR      T4645  ; 進左開夾不在位置上延遲
      ANB
      OUT     M4645  ; 進料左側開夾不在位置上
5332  LD      L207  ; 伺服馬達不在位置上異常  Enable
      AND     T1000  ; 開機延遲
      MPS
      ANI     X0A16  ; #07 AXIS Busy
      ANI     L1730  ; 進右開爪位置01  操作側
      ANI     L1731  ; 進右開爪位置02  出料側
      ANI     L1732  ; 進右開爪位置03
      ANI     L1733  ; 進右開爪位置04
      ANI     L1734  ; 進右開爪位置05
      OUT     T4646 K10  ; 進右開夾不在位置上延遲
      MPP
      LD      M4646  ; 進料右側開夾不在位置上
      ANI     L4034  ; 回流段  異常復歸
      OR      T4646  ; 進右開夾不在位置上延遲
      ANB
      OUT     M4646  ; 進料右側開夾不在位置上
5351  LD      L207  ; 伺服馬達不在位置上異常  Enable
      AND     T1000  ; 開機延遲
      MPS
      ANI     X0A17  ; #08 AXIS Busy
      ANI     L2130  ; 分流前取框位置01  出料側
      ANI     L2131  ; 分流前取框位置02進料側
      OUT     T4647 K10  ; 分流前取框不在位置上延遲
      MPP
      LD      M4647  ; 分流前取框不在位置上
      ANI     L4032  ; 爐體段  異常復歸
      OR      T4647  ; 分流前取框不在位置上延遲
      ANB
      OUT     M4647  ; 分流前取框不在位置上
5367  LD      M7601  ; Run Off
      AND     L207  ; 伺服馬達不在位置上異常  Enable
      AND     T1000  ; 開機延遲
      MPS
      ANI     X0A18  ; #09 AXIS Busy
      ANI     L3530  ; 出板牙插移載位置01
      ANI     L3531  ; 出板牙插移載位置02
      OUT     T4648 K10  ; 出板牙插不在位置上延遲
      MPP
      LD      M4648  ; 出板牙插不在位置上
      ANI     L4033  ; 出料段  異常復歸
      OR      T4648  ; 出板牙插不在位置上延遲
      ANB
      OUT     M4648  ; 出板牙插不在位置上
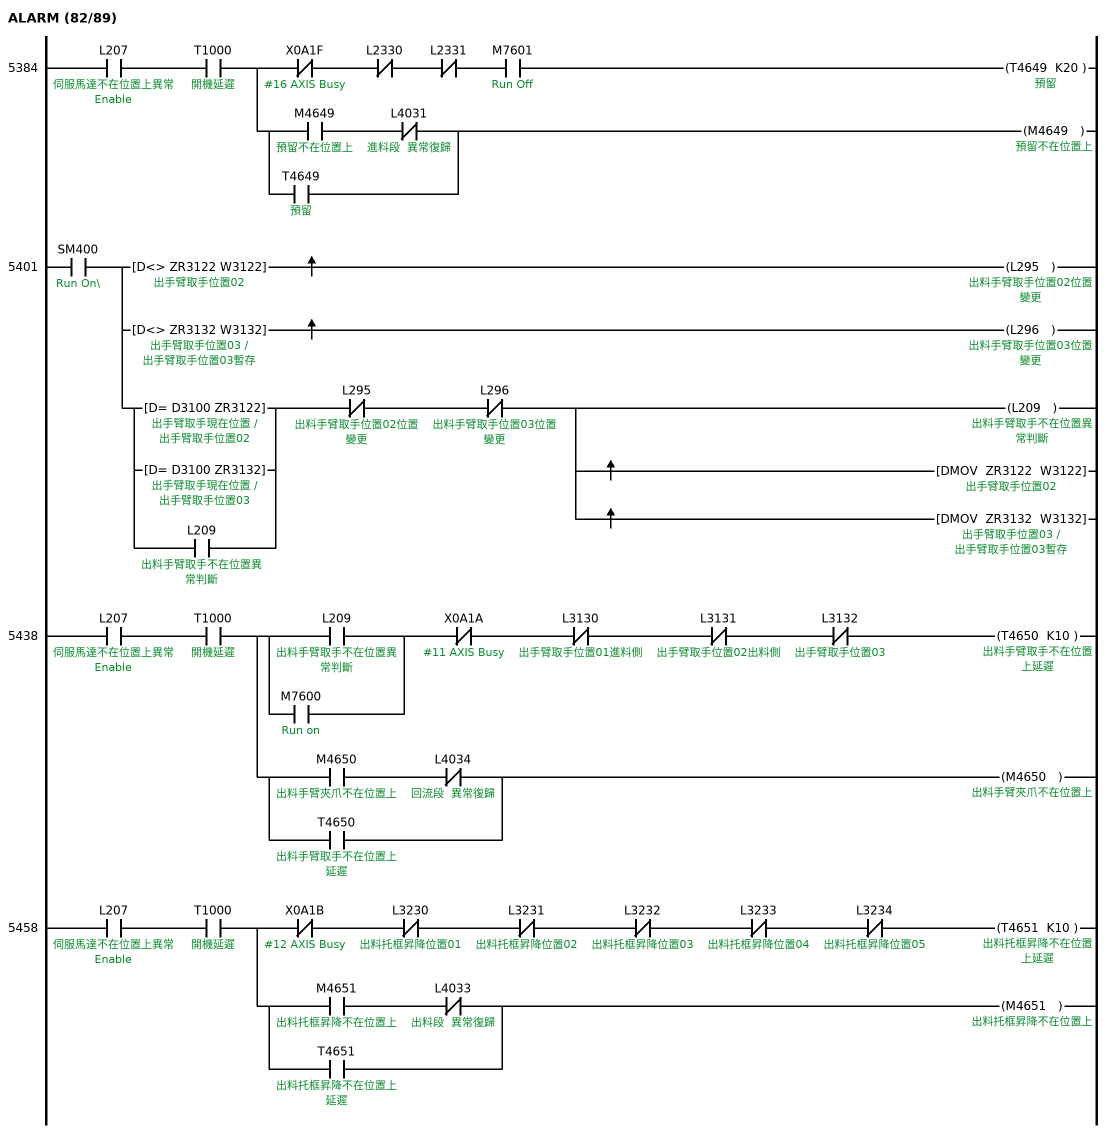
5384  LD      L207  ; 伺服馬達不在位置上異常  Enable
      AND     T1000  ; 開機延遲
      MPS
      ANI     X0A1F  ; #16 AXIS Busy
      ANI     L2330
      ANI     L2331
      AND     M7601  ; Run Off
      OUT     T4649 K20  ; 預留
      MPP
      LD      M4649  ; 預留不在位置上
      ANI     L4031  ; 進料段  異常復歸
      OR      T4649  ; 預留
      ANB
      OUT     M4649  ; 預留不在位置上
5401  LD      SM400  ; Run On\
      MPS
      ANDD<>  ZR3122 W3122  ; 出手臂取手位置02
      MEP
      OUT     L295  ; 出料手臂取手位置02位置變更
      MRD
      ANDD<>  ZR3132 W3132  ; 出手臂取手位置03 / 出手臂取手位置03暫存
      MEP
      OUT     L296  ; 出料手臂取手位置03位置變更
      MPP
      LDD=    D3100 ZR3122  ; 出手臂取手現在位置 / 出手臂取手位置02
      ORD=    D3100 ZR3132  ; 出手臂取手現在位置 / 出手臂取手位置03
      OR      L209  ; 出料手臂取手不在位置異常判斷
      ANB
      ANI     L295  ; 出料手臂取手位置02位置變更
      ANI     L296  ; 出料手臂取手位置03位置變更
      OUT     L209  ; 出料手臂取手不在位置異常判斷
      MPS
      MEP
      DMOV    ZR3122 W3122
      MPP
      MEP
      DMOV    ZR3132 W3132
5438  LD      L207  ; 伺服馬達不在位置上異常  Enable
      AND     T1000  ; 開機延遲
      MPS
      LD      L209  ; 出料手臂取手不在位置異常判斷
      OR      M7600  ; Run on
      ANB
      ANI     X0A1A  ; #11 AXIS Busy
      ANI     L3130  ; 出手臂取手位置01進料側
      ANI     L3131  ; 出手臂取手位置02出料側
      ANI     L3132  ; 出手臂取手位置03
      OUT     T4650 K10  ; 出料手臂取手不在位置上延遲
      MPP
      LD      M4650  ; 出料手臂夾爪不在位置上
      ANI     L4034  ; 回流段  異常復歸
      OR      T4650  ; 出料手臂取手不在位置上延遲
      ANB
      OUT     M4650  ; 出料手臂夾爪不在位置上
5458  LD      L207  ; 伺服馬達不在位置上異常  Enable
      AND     T1000  ; 開機延遲
      MPS
      ANI     X0A1B  ; #12 AXIS Busy
      ANI     L3230  ; 出料托框昇降位置01
      ANI     L3231  ; 出料托框昇降位置02
      ANI     L3232  ; 出料托框昇降位置03
      ANI     L3233  ; 出料托框昇降位置04
      ANI     L3234  ; 出料托框昇降位置05
      OUT     T4651 K10  ; 出料托框昇降不在位置上延遲
      MPP
      LD      M4651  ; 出料托框昇降不在位置上
      ANI     L4033  ; 出料段  異常復歸
      OR      T4651  ; 出料托框昇降不在位置上延遲
      ANB
      OUT     M4651  ; 出料托框昇降不在位置上
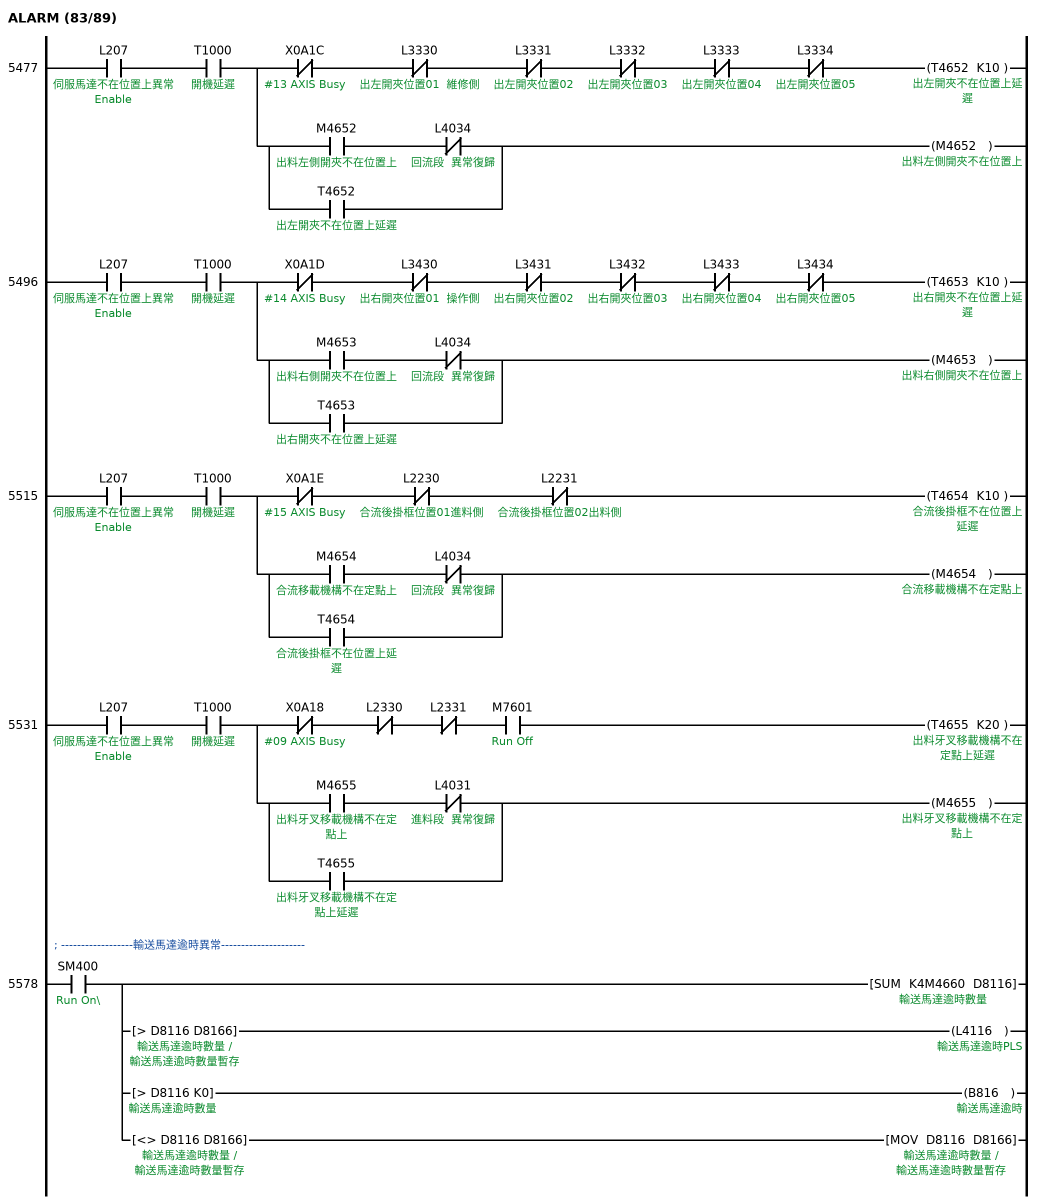
5477  LD      L207  ; 伺服馬達不在位置上異常  Enable
      AND     T1000  ; 開機延遲
      MPS
      ANI     X0A1C  ; #13 AXIS Busy
      ANI     L3330  ; 出左開夾位置01  維修側
      ANI     L3331  ; 出左開夾位置02
      ANI     L3332  ; 出左開夾位置03
      ANI     L3333  ; 出左開夾位置04
      ANI     L3334  ; 出左開夾位置05
      OUT     T4652 K10  ; 出左開夾不在位置上延遲
      MPP
      LD      M4652  ; 出料左側開夾不在位置上
      ANI     L4034  ; 回流段  異常復歸
      OR      T4652  ; 出左開夾不在位置上延遲
      ANB
      OUT     M4652  ; 出料左側開夾不在位置上
5496  LD      L207  ; 伺服馬達不在位置上異常  Enable
      AND     T1000  ; 開機延遲
      MPS
      ANI     X0A1D  ; #14 AXIS Busy
      ANI     L3430  ; 出右開夾位置01  操作側
      ANI     L3431  ; 出右開夾位置02
      ANI     L3432  ; 出右開夾位置03
      ANI     L3433  ; 出右開夾位置04
      ANI     L3434  ; 出右開夾位置05
      OUT     T4653 K10  ; 出右開夾不在位置上延遲
      MPP
      LD      M4653  ; 出料右側開夾不在位置上
      ANI     L4034  ; 回流段  異常復歸
      OR      T4653  ; 出右開夾不在位置上延遲
      ANB
      OUT     M4653  ; 出料右側開夾不在位置上
5515  LD      L207  ; 伺服馬達不在位置上異常  Enable
      AND     T1000  ; 開機延遲
      MPS
      ANI     X0A1E  ; #15 AXIS Busy
      ANI     L2230  ; 合流後掛框位置01進料側
      ANI     L2231  ; 合流後掛框位置02出料側
      OUT     T4654 K10  ; 合流後掛框不在位置上延遲
      MPP
      LD      M4654  ; 合流移載機構不在定點上
      ANI     L4034  ; 回流段  異常復歸
      OR      T4654  ; 合流後掛框不在位置上延遲
      ANB
      OUT     M4654  ; 合流移載機構不在定點上
5531  LD      L207  ; 伺服馬達不在位置上異常  Enable
      AND     T1000  ; 開機延遲
      MPS
      ANI     X0A18  ; #09 AXIS Busy
      ANI     L2330
      ANI     L2331
      AND     M7601  ; Run Off
      OUT     T4655 K20  ; 出料牙叉移載機構不在定點上延遲
      MPP
      LD      M4655  ; 出料牙叉移載機構不在定點上
      ANI     L4031  ; 進料段  異常復歸
      OR      T4655  ; 出料牙叉移載機構不在定點上延遲
      ANB
      OUT     M4655  ; 出料牙叉移載機構不在定點上
; ------------------輸送馬達逾時異常---------------------
5578  LD      SM400  ; Run On\
      SUM     K4M4660 D8116  ; 進料整板動作逾時 / 輸送馬達逾時數量
      MPS
      AND>    D8116 D8166  ; 輸送馬達逾時數量 / 輸送馬達逾時數量暫存
      OUT     L4116  ; 輸送馬達逾時PLS
      MRD
      AND>    D8116 K0  ; 輸送馬達逾時數量
      OUT     B816  ; 輸送馬達逾時
      MPP
      AND<>   D8116 D8166  ; 輸送馬達逾時數量 / 輸送馬達逾時數量暫存
      MOV     D8116 D8166
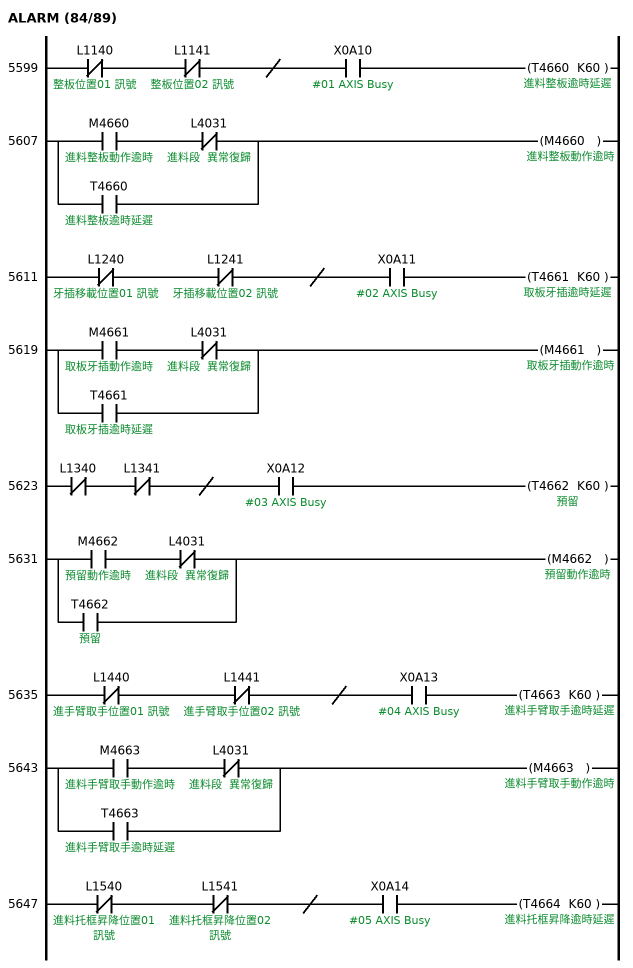
5599  LDI     L1140  ; 整板位置01 訊號
      ANI     L1141  ; 整板位置02 訊號
      INV
      AND     X0A10  ; #01 AXIS Busy
      OUT     T4660 K60  ; 進料整板逾時延遲
5607  LD      M4660  ; 進料整板動作逾時
      ANI     L4031  ; 進料段  異常復歸
      OR      T4660  ; 進料整板逾時延遲
      OUT     M4660  ; 進料整板動作逾時
5611  LDI     L1240  ; 牙插移載位置01 訊號
      ANI     L1241  ; 牙插移載位置02 訊號
      INV
      AND     X0A11  ; #02 AXIS Busy
      OUT     T4661 K60  ; 取板牙插逾時延遲
5619  LD      M4661  ; 取板牙插動作逾時
      ANI     L4031  ; 進料段  異常復歸
      OR      T4661  ; 取板牙插逾時延遲
      OUT     M4661  ; 取板牙插動作逾時
5623  LDI     L1340
      ANI     L1341
      INV
      AND     X0A12  ; #03 AXIS Busy
      OUT     T4662 K60  ; 預留
5631  LD      M4662  ; 預留動作逾時
      ANI     L4031  ; 進料段  異常復歸
      OR      T4662  ; 預留
      OUT     M4662  ; 預留動作逾時
5635  LDI     L1440  ; 進手臂取手位置01 訊號
      ANI     L1441  ; 進手臂取手位置02 訊號
      INV
      AND     X0A13  ; #04 AXIS Busy
      OUT     T4663 K60  ; 進料手臂取手逾時延遲
5643  LD      M4663  ; 進料手臂取手動作逾時
      ANI     L4031  ; 進料段  異常復歸
      OR      T4663  ; 進料手臂取手逾時延遲
      OUT     M4663  ; 進料手臂取手動作逾時
5647  LDI     L1540  ; 進料托框昇降位置01 訊號
      ANI     L1541  ; 進料托框昇降位置02 訊號
      INV
      AND     X0A14  ; #05 AXIS Busy
      OUT     T4664 K60  ; 進料托框昇降逾時延遲
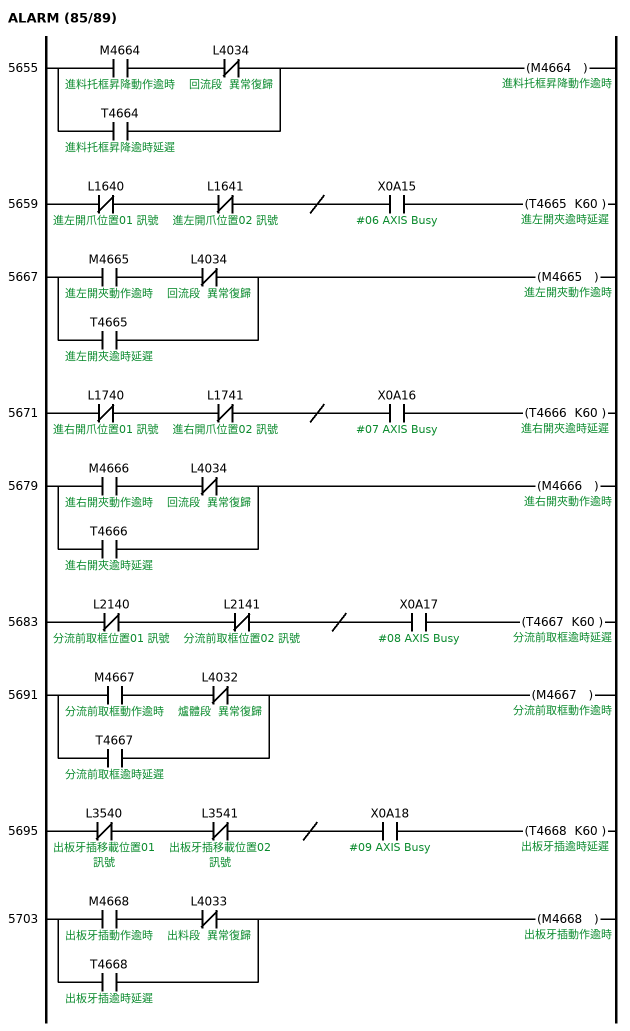
5655  LD      M4664  ; 進料托框昇降動作逾時
      ANI     L4034  ; 回流段  異常復歸
      OR      T4664  ; 進料托框昇降逾時延遲
      OUT     M4664  ; 進料托框昇降動作逾時
5659  LDI     L1640  ; 進左開爪位置01 訊號
      ANI     L1641  ; 進左開爪位置02 訊號
      INV
      AND     X0A15  ; #06 AXIS Busy
      OUT     T4665 K60  ; 進左開夾逾時延遲
5667  LD      M4665  ; 進左開夾動作逾時
      ANI     L4034  ; 回流段  異常復歸
      OR      T4665  ; 進左開夾逾時延遲
      OUT     M4665  ; 進左開夾動作逾時
5671  LDI     L1740  ; 進右開爪位置01 訊號
      ANI     L1741  ; 進右開爪位置02 訊號
      INV
      AND     X0A16  ; #07 AXIS Busy
      OUT     T4666 K60  ; 進右開夾逾時延遲
5679  LD      M4666  ; 進右開夾動作逾時
      ANI     L4034  ; 回流段  異常復歸
      OR      T4666  ; 進右開夾逾時延遲
      OUT     M4666  ; 進右開夾動作逾時
5683  LDI     L2140  ; 分流前取框位置01 訊號
      ANI     L2141  ; 分流前取框位置02 訊號
      INV
      AND     X0A17  ; #08 AXIS Busy
      OUT     T4667 K60  ; 分流前取框逾時延遲
5691  LD      M4667  ; 分流前取框動作逾時
      ANI     L4032  ; 爐體段  異常復歸
      OR      T4667  ; 分流前取框逾時延遲
      OUT     M4667  ; 分流前取框動作逾時
5695  LDI     L3540  ; 出板牙插移載位置01 訊號
      ANI     L3541  ; 出板牙插移載位置02 訊號
      INV
      AND     X0A18  ; #09 AXIS Busy
      OUT     T4668 K60  ; 出板牙插逾時延遲
5703  LD      M4668  ; 出板牙插動作逾時
      ANI     L4033  ; 出料段  異常復歸
      OR      T4668  ; 出板牙插逾時延遲
      OUT     M4668  ; 出板牙插動作逾時
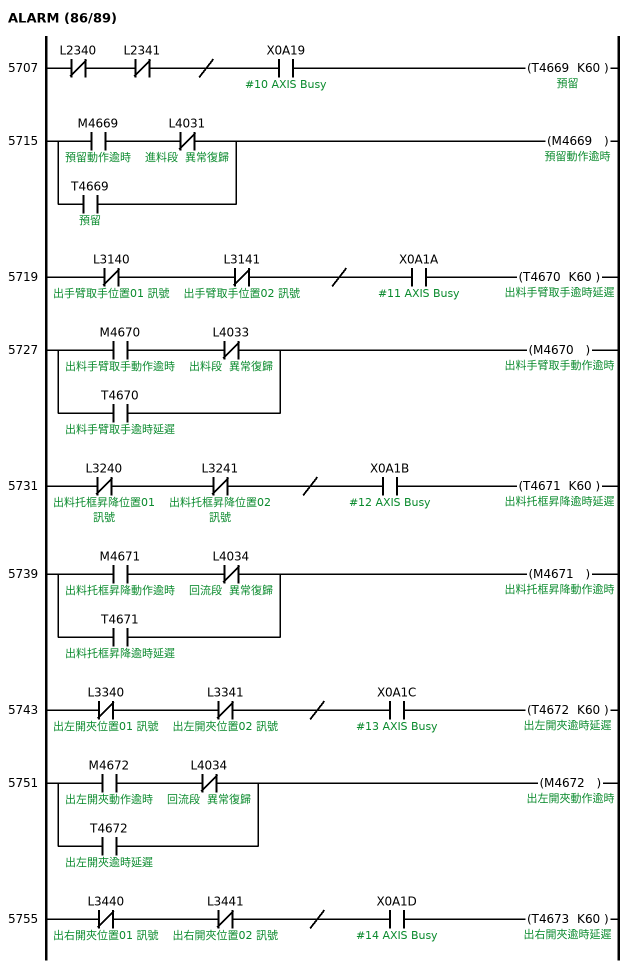
5707  LDI     L2340
      ANI     L2341
      INV
      AND     X0A19  ; #10 AXIS Busy
      OUT     T4669 K60  ; 預留
5715  LD      M4669  ; 預留動作逾時
      ANI     L4031  ; 進料段  異常復歸
      OR      T4669  ; 預留
      OUT     M4669  ; 預留動作逾時
5719  LDI     L3140  ; 出手臂取手位置01 訊號
      ANI     L3141  ; 出手臂取手位置02 訊號
      INV
      AND     X0A1A  ; #11 AXIS Busy
      OUT     T4670 K60  ; 出料手臂取手逾時延遲
5727  LD      M4670  ; 出料手臂取手動作逾時
      ANI     L4033  ; 出料段  異常復歸
      OR      T4670  ; 出料手臂取手逾時延遲
      OUT     M4670  ; 出料手臂取手動作逾時
5731  LDI     L3240  ; 出料托框昇降位置01 訊號
      ANI     L3241  ; 出料托框昇降位置02 訊號
      INV
      AND     X0A1B  ; #12 AXIS Busy
      OUT     T4671 K60  ; 出料托框昇降逾時延遲
5739  LD      M4671  ; 出料托框昇降動作逾時
      ANI     L4034  ; 回流段  異常復歸
      OR      T4671  ; 出料托框昇降逾時延遲
      OUT     M4671  ; 出料托框昇降動作逾時
5743  LDI     L3340  ; 出左開夾位置01 訊號
      ANI     L3341  ; 出左開夾位置02 訊號
      INV
      AND     X0A1C  ; #13 AXIS Busy
      OUT     T4672 K60  ; 出左開夾逾時延遲
5751  LD      M4672  ; 出左開夾動作逾時
      ANI     L4034  ; 回流段  異常復歸
      OR      T4672  ; 出左開夾逾時延遲
      OUT     M4672  ; 出左開夾動作逾時
5755  LDI     L3440  ; 出右開夾位置01 訊號
      ANI     L3441  ; 出右開夾位置02 訊號
      INV
      AND     X0A1D  ; #14 AXIS Busy
      OUT     T4673 K60  ; 出右開夾逾時延遲
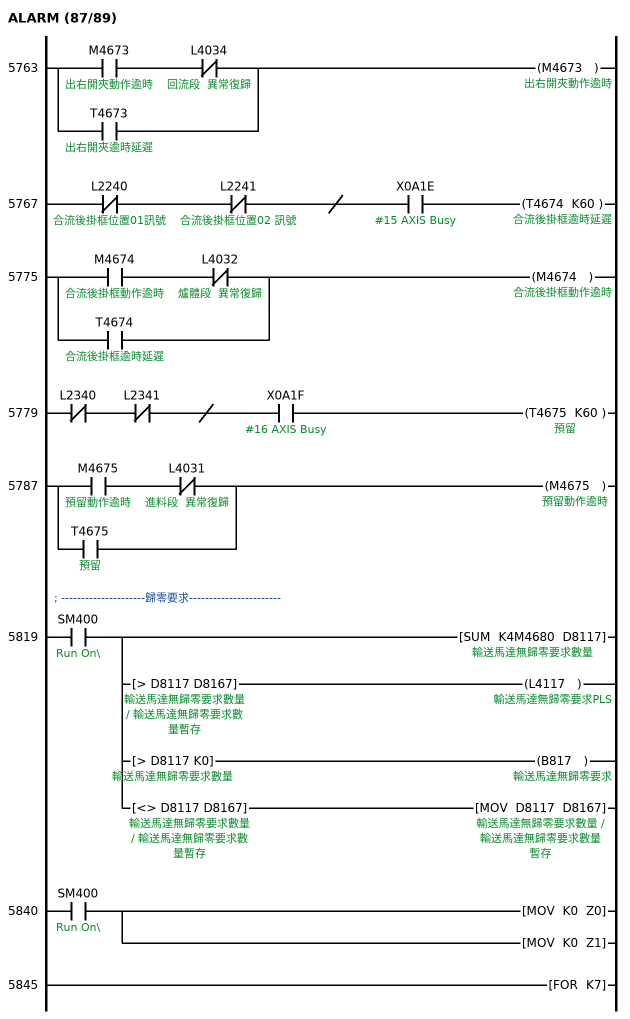
5763  LD      M4673  ; 出右開夾動作逾時
      ANI     L4034  ; 回流段  異常復歸
      OR      T4673  ; 出右開夾逾時延遲
      OUT     M4673  ; 出右開夾動作逾時
5767  LDI     L2240  ; 合流後掛框位置01訊號
      ANI     L2241  ; 合流後掛框位置02 訊號
      INV
      AND     X0A1E  ; #15 AXIS Busy
      OUT     T4674 K60  ; 合流後掛框逾時延遲
5775  LD      M4674  ; 合流後掛框動作逾時
      ANI     L4032  ; 爐體段  異常復歸
      OR      T4674  ; 合流後掛框逾時延遲
      OUT     M4674  ; 合流後掛框動作逾時
5779  LDI     L2340
      ANI     L2341
      INV
      AND     X0A1F  ; #16 AXIS Busy
      OUT     T4675 K60  ; 預留
5787  LD      M4675  ; 預留動作逾時
      ANI     L4031  ; 進料段  異常復歸
      OR      T4675  ; 預留
      OUT     M4675  ; 預留動作逾時
; ---------------------歸零要求-----------------------
5819  LD      SM400  ; Run On\
      SUM     K4M4680 D8117  ; 進料整板歸零要求異常 / 輸送馬達無歸零要求數量
      MPS
      AND>    D8117 D8167  ; 輸送馬達無歸零要求數量 / 輸送馬達無歸零要求數量暫存
      OUT     L4117  ; 輸送馬達無歸零要求PLS
      MRD
      AND>    D8117 K0  ; 輸送馬達無歸零要求數量
      OUT     B817  ; 輸送馬達無歸零要求
      MPP
      AND<>   D8117 D8167  ; 輸送馬達無歸零要求數量 / 輸送馬達無歸零要求數量暫存
      MOV     D8117 D8167
5840  LD      SM400  ; Run On\
      MOV     K0 Z0
      MOV     K0 Z1
5845  FOR     K7
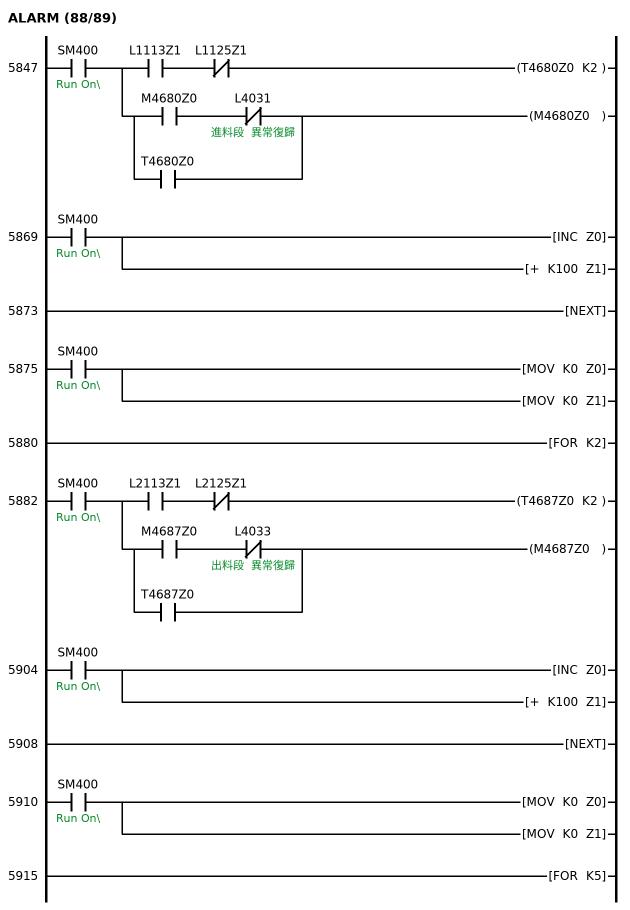
5847  LD      SM400  ; Run On\
      MPS
      AND     L1113Z1
      ANI     L1125Z1
      OUT     T4680Z0 K2
      MPP
      LD      M4680Z0
      ANI     L4031  ; 進料段  異常復歸
      OR      T4680Z0
      ANB
      OUT     M4680Z0
5869  LD      SM400  ; Run On\
      INC     Z0
      +       K100 Z1
5873  NEXT
5875  LD      SM400  ; Run On\
      MOV     K0 Z0
      MOV     K0 Z1
5880  FOR     K2
5882  LD      SM400  ; Run On\
      MPS
      AND     L2113Z1
      ANI     L2125Z1
      OUT     T4687Z0 K2
      MPP
      LD      M4687Z0
      ANI     L4033  ; 出料段  異常復歸
      OR      T4687Z0
      ANB
      OUT     M4687Z0
5904  LD      SM400  ; Run On\
      INC     Z0
      +       K100 Z1
5908  NEXT
5910  LD      SM400  ; Run On\
      MOV     K0 Z0
      MOV     K0 Z1
5915  FOR     K5
